(* PLC project Generated.project, CODESYS CODESYS V3.5 SP19 Patch 1 *)
(* stored: creationDateTime 2026-09-03T14:40:09.654789, modificationDateTime 2026-09-03T14:40:09.654789 *)

(* ═══════════════════════════════════════════════════════════════ ⚙️ ST_MachineHomingCfg — Réglages IHM du cycle de référencement machine ─────────────────────────────────────────────────────────────── 🎯 Mise en service. Les réglages géométriques (positions capteur, offsets benne) restent portés par GVL_PERSISTENT (_WinchM1CfgPersist / _BucketCfgPersist). 💾 Ponté vers persist (_MachineHomingCfgPersist) via FB_CfgPersistBridge_MachineHomingCfg. ═══════════════════════════════════════════════════════════════ *)
TYPE ST_MachineHomingCfg : STRUCT
  ForceStepTarget : INT := 0;  (* 🔧 Step GRAFCET cible du forçage (0=HX0 .. 9=HXF), borné côté FB *)
  Initialized : BOOL := FALSE;  (* 🚦 flag restauration boot *)
END_STRUCT;
END_TYPE
